TEXTLIST TL_Lang
  0 = 'English' | EN\: 'English' | EN: 'English' | PL: 'Angielski' | PL\: 'Angielski'
  1 = 'Polish' | EN\: 'Polish' | EN: 'Polish' | PL: 'Polski' | PL\: 'Polski'
   = ''
END_TEXTLIST

(* stored: Version 1.1.0.1, ProductVersion 3.1.4022.6
   TextList TL_Lang: Id {97a347aa-12ba-434c-b88f-18e1bc16df89} *)
